(* Logix 5000 project; controller Receptivo vendor 1 type 14 code 106 rev 30.11; software revision 30.00; part 10 of 10 *)
(* tags used below, declared in another part *)
   CHASSIS_CURRENT : INT;
   CONTROLLER_STATUS : DINT;
   CPUdiag_FlashingGreen : BOOL;
   CPUdiag_FlashingRed : BOOL;
   CPUdiag_LEDStatus : DINT;
   CPUdiag_Major : MajorFaultBits;
   CPUdiag_MajorEvents : INT;
   CPUdiag_MajorFaultBits : DINT;
   CPUdiag_Minor : MinorFaultBits;
   CPUdiag_MinorEvents : INT;
   CPUdiag_MinorFaultBits : DINT;
   CPUdiag_SolidGreen : BOOL;
   CPUdiag_StatusMasked : INT;
   CPUdiag_StatusRaw : INT;
   INDEX : INT;
   IO_TREE_NO_OK : BOOL;
   IO_TREE_OK : DINT;
   MINOR_FAULTS : DINT;
   MODULE_MASK : DINT[10,17];
   MODULE_STATUS : DINT[10,17];
   Printer_Zebra_OK : BOOL;
   Timer1 : TIMER;
   ACTIVE_SLOT : DINT[10];
   Autonegotiation_Fallo : BOOL;
   Autonegotiation_OK : BOOL;
   Autonegotiation_Start : BOOL;
   AutoNegotiation_Status : SINT;
   CLOCK : DINT[7];
   Ethernet_Duplex_OK : BOOL;
   Ethernet_Duplex_State : ALIAS FOR Ethernet_Module_Status.1;
   Ethernet_Hardware_Mal : BOOL;
   Ethernet_Hardware_Status : ALIAS FOR Ethernet_Module_Status.6;
   Ethernet_Link_State : ALIAS FOR Ethernet_Module_Status.0;
   Ethernet_Module_Status : DINT;
   ETHERNET_STATUS : Ethernet_Status;
   FLASH_TIMERS : TIMER[2];
   FORCE_STATUS : DINT;
   Get_Ethernet_Module_Link_Status : MESSAGE;
   Hardy_Basculas_Net_OK : BOOL;
   KEY_SWITCH_REM_RUN : BOOL;
   KEY_SWITCH_RUN : BOOL;
   MODULE_FAULT_STATUS : DINT[10];
   Modulo_Ethernet_Mal : BOOL;
   Prueba : UDT_COLA[3];
   SYSTEM_STATUS_COMPLETE : BOOL;
   Velocidad_Modo_Forzado : BOOL;
(* SYSTEM_STATUS, continued *)

ROUTINE Ethernet_Module_Status   (* ladder *)
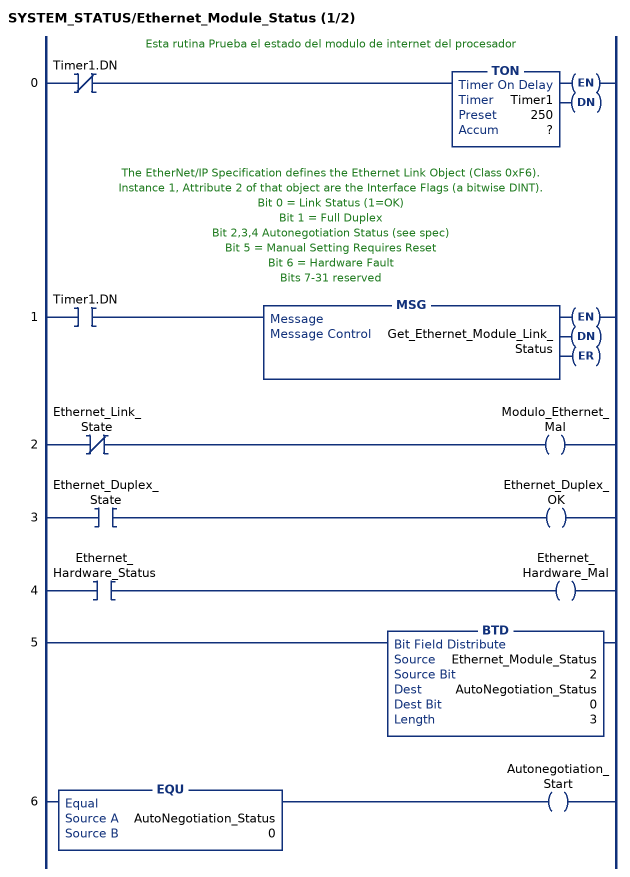
   // Esta rutina Prueba el estado del modulo de internet del procesador
   0: XIO(Timer1.DN)TON(Timer1,?,?);
   // The EtherNet/IP Specification defines the Ethernet Link Object (Class 0xF6).
   // Instance 1, Attribute 2 of that object are the Interface Flags (a bitwise DINT).
   // Bit 0 = Link Status (1=OK)
   // Bit 1 = Full Duplex
   // Bit 2,3,4 Autonegotiation Status (see spec)
   // Bit 5 = Manual Setting Requires Reset
   // Bit 6 = Hardware Fault
   // Bits 7-31 reserved
   1: XIC(Timer1.DN)MSG(Get_Ethernet_Module_Link_Status);
   2: XIO(Ethernet_Link_State)OTE(Modulo_Ethernet_Mal);
   3: XIC(Ethernet_Duplex_State)OTE(Ethernet_Duplex_OK);
   4: XIC(Ethernet_Hardware_Status)OTE(Ethernet_Hardware_Mal);
   5: BTD(Ethernet_Module_Status,2,AutoNegotiation_Status,0,3);
   6: EQU(AutoNegotiation_Status,0)OTE(Autonegotiation_Start);
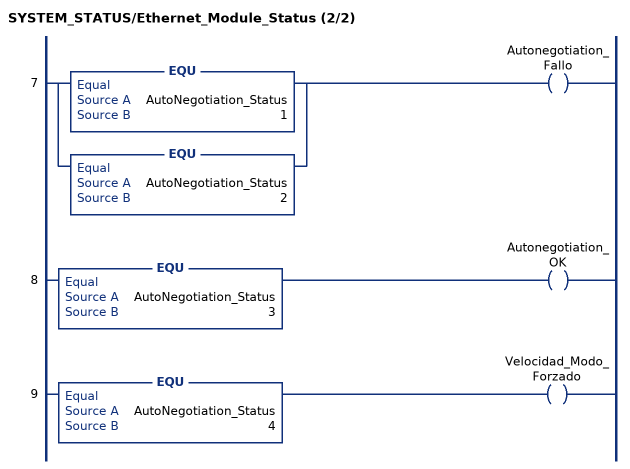
   7: [EQU(AutoNegotiation_Status,1) ,EQU(AutoNegotiation_Status,2) ]OTE(Autonegotiation_Fallo);
   8: EQU(AutoNegotiation_Status,3)OTE(Autonegotiation_OK);
   9: EQU(AutoNegotiation_Status,4)OTE(Velocidad_Modo_Forzado);
END_ROUTINE

ROUTINE ETHERNET_STATUS   (* ladder *)
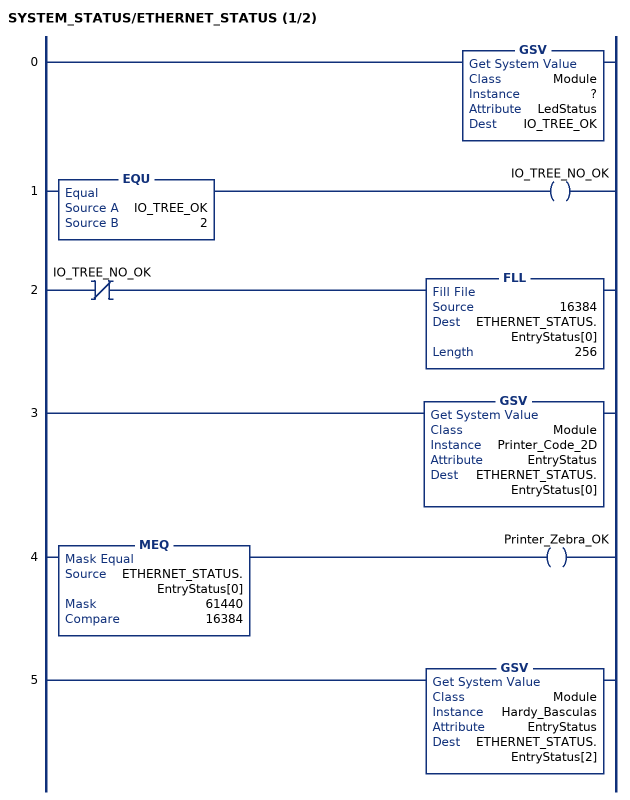
   0: GSV(Module,?,LedStatus,IO_TREE_OK);
   1: EQU(IO_TREE_OK,2)OTE(IO_TREE_NO_OK);
   2: XIO(IO_TREE_NO_OK)FLL(16384,ETHERNET_STATUS.EntryStatus[0],256);
   3: GSV(Module,Printer_Code_2D,EntryStatus,ETHERNET_STATUS.EntryStatus[0]);
   4: MEQ(ETHERNET_STATUS.EntryStatus[0],61440,16384)OTE(Printer_Zebra_OK);
   5: GSV(Module,Hardy_Basculas,EntryStatus,ETHERNET_STATUS.EntryStatus[2]);
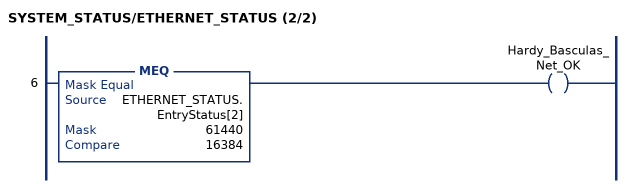
   6: MEQ(ETHERNET_STATUS.EntryStatus[2],61440,16384)OTE(Hardy_Basculas_Net_OK);
END_ROUTINE

ROUTINE GET_CONTROLLER_STATUS   (* ladder *)
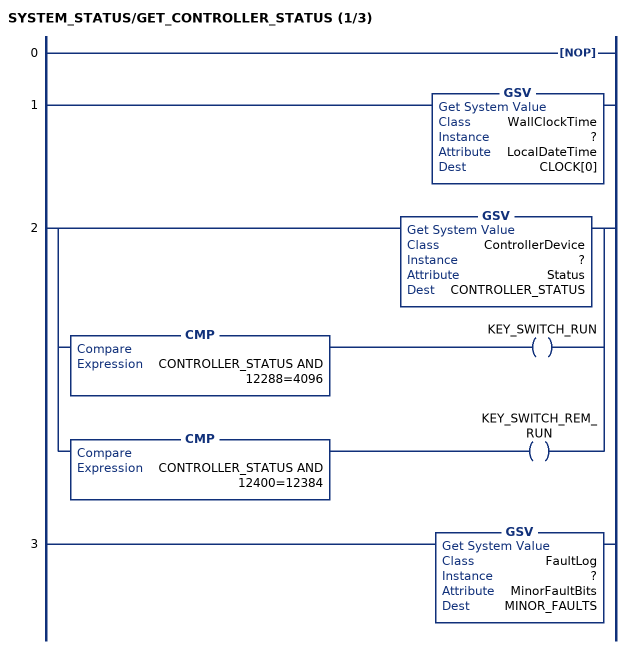
   0: NOP();
   1: GSV(WallClockTime,?,LocalDateTime,CLOCK[0]);
   2: [GSV(ControllerDevice,?,Status,CONTROLLER_STATUS) ,CMP(CONTROLLER_STATUS AND 12288=4096) OTE(KEY_SWITCH_RUN) ,CMP(CONTROLLER_STATUS AND 12400=12384) OTE(KEY_SWITCH_REM_RUN) ];
   3: GSV(FaultLog,?,MinorFaultBits,MINOR_FAULTS);
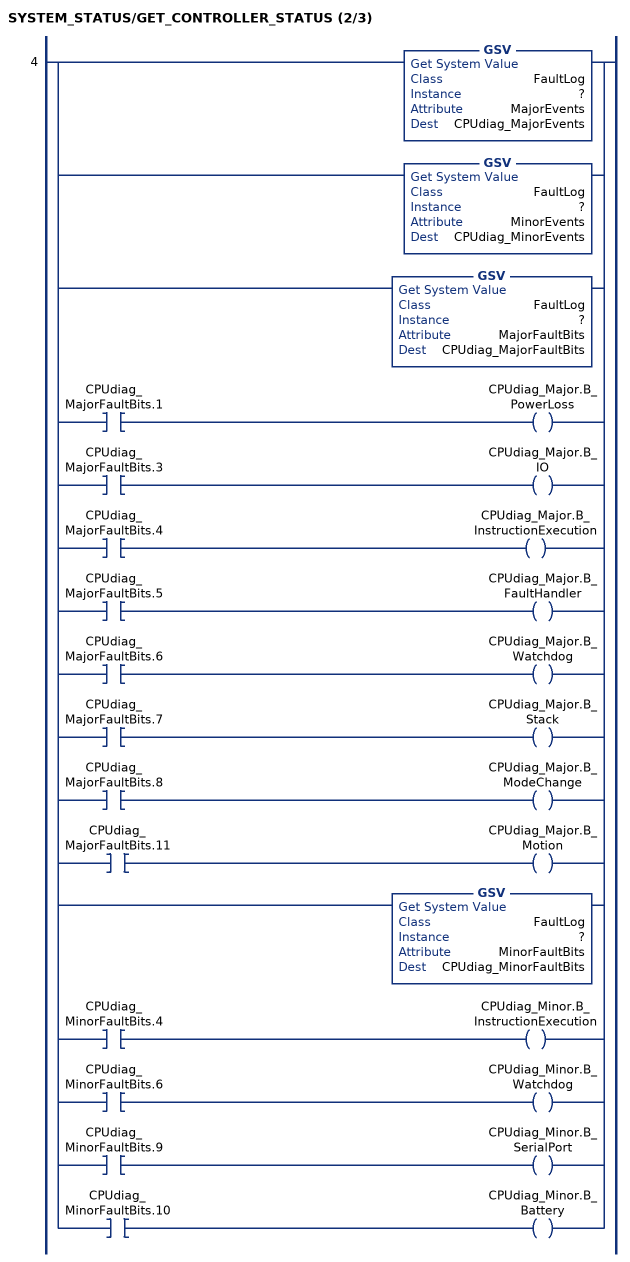
   4: [GSV(FaultLog,?,MajorEvents,CPUdiag_MajorEvents) ,GSV(FaultLog,?,MinorEvents,CPUdiag_MinorEvents) ,GSV(FaultLog,?,MajorFaultBits,CPUdiag_MajorFaultBits) ,XIC(CPUdiag_MajorFaultBits.1) OTE(CPUdiag_Major.B_PowerLoss) ,XIC(CPUdiag_MajorFaultBits.3) OTE(CPUdiag_Major.B_IO) ,XIC(CPUdiag_MajorFaultBits.4) OTE(CPUdiag_Major.B_InstructionExecution) ,XIC(CPUdiag_MajorFaultBits.5) OTE(CPUdiag_Major.B_FaultHandler) ,XIC(CPUdiag_MajorFaultBits.6) OTE(CPUdiag_Major.B_Watchdog) ,XIC(CPUdiag_MajorFaultBits.7) OTE(CPUdiag_Major.B_Stack) ,XIC(CPUdiag_MajorFaultBits.8) OTE(CPUdiag_Major.B_ModeChange) ,XIC(CPUdiag_MajorFaultBits.11) OTE(CPUdiag_Major.B_Motion) ,GSV(FaultLog,?,MinorFaultBits,CPUdiag_MinorFaultBits) ,XIC(CPUdiag_MinorFaultBits.4) OTE(CPUdiag_Minor.B_InstructionExecution) ,XIC(CPUdiag_MinorFaultBits.6) OTE(CPUdiag_Minor.B_Watchdog) ,XIC(CPUdiag_MinorFaultBits.9) OTE(CPUdiag_Minor.B_SerialPort) ,XIC(CPUdiag_MinorFaultBits.10) OTE(CPUdiag_Minor.B_Battery) ];
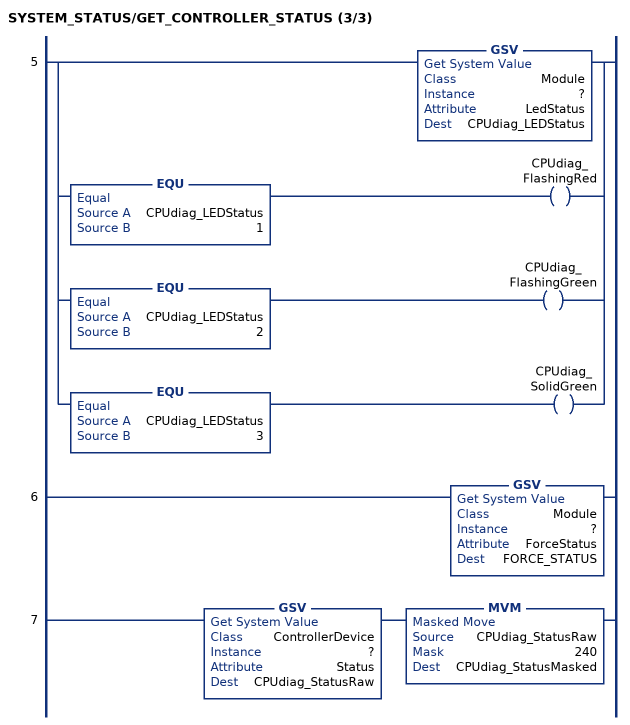
   5: [GSV(Module,?,LedStatus,CPUdiag_LEDStatus) ,EQU(CPUdiag_LEDStatus,1) OTE(CPUdiag_FlashingRed) ,EQU(CPUdiag_LEDStatus,2) OTE(CPUdiag_FlashingGreen) ,EQU(CPUdiag_LEDStatus,3) OTE(CPUdiag_SolidGreen) ];
   6: GSV(Module,?,ForceStatus,FORCE_STATUS);
   7: GSV(ControllerDevice,?,Status,CPUdiag_StatusRaw)MVM(CPUdiag_StatusRaw,240,CPUdiag_StatusMasked);
END_ROUTINE

ROUTINE GET_MODULE_STATUS   (* ladder *)
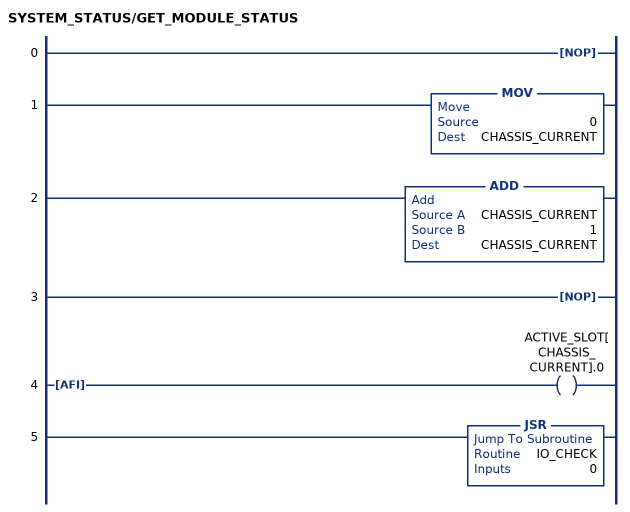
   0: NOP();
   1: MOV(0,CHASSIS_CURRENT);
   2: ADD(CHASSIS_CURRENT,1,CHASSIS_CURRENT);
   3: NOP();
   4: AFI()OTE(ACTIVE_SLOT[CHASSIS_CURRENT].0);
   5: JSR(IO_CHECK,0);
END_ROUTINE

ROUTINE IO_CHECK   (* ladder *)
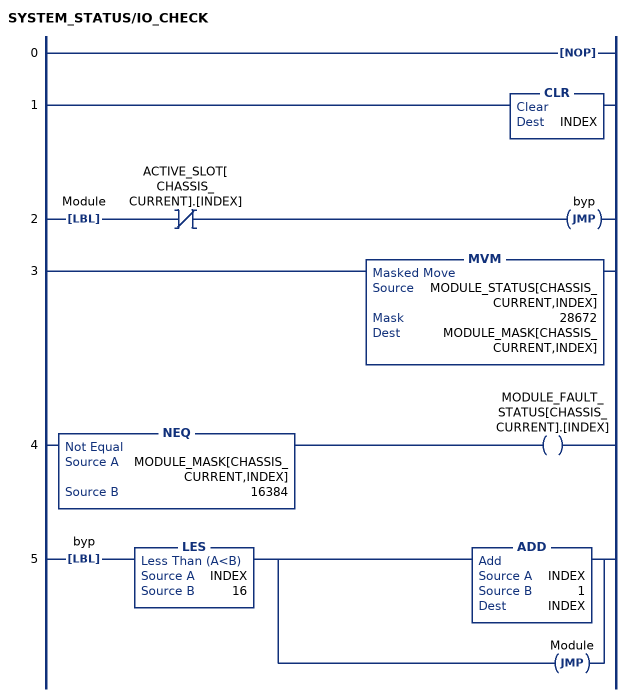
   0: NOP();
   1: CLR(INDEX);
   2: LBL(Module)XIO(ACTIVE_SLOT[CHASSIS_CURRENT].[INDEX])JMP(byp);
   3: MVM(MODULE_STATUS[CHASSIS_CURRENT,INDEX],28672,MODULE_MASK[CHASSIS_CURRENT,INDEX]);
   4: NEQ(MODULE_MASK[CHASSIS_CURRENT,INDEX],16384)OTE(MODULE_FAULT_STATUS[CHASSIS_CURRENT].[INDEX]);
   5: LBL(byp)LES(INDEX,16)[ADD(INDEX,1,INDEX) ,JMP(Module) ];
END_ROUTINE

ROUTINE MAIN   (* ladder *)
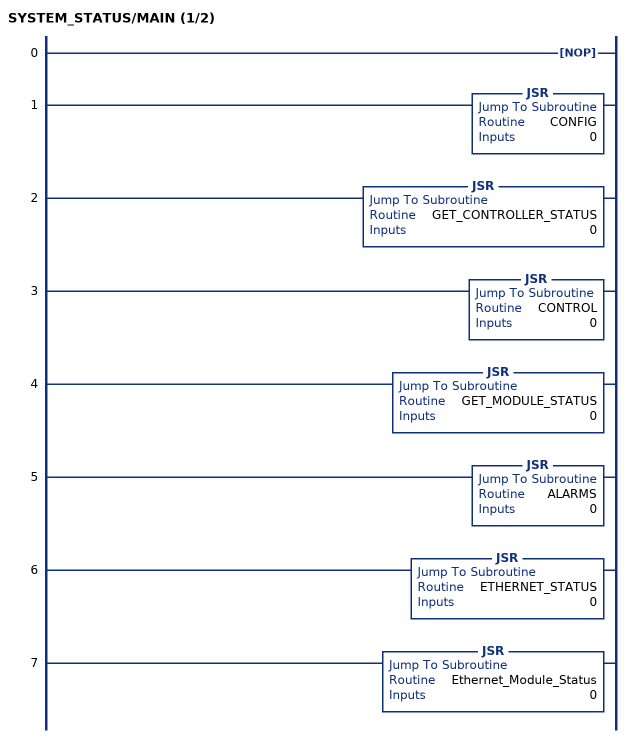
   0: NOP();
   1: JSR(CONFIG,0);
   2: JSR(GET_CONTROLLER_STATUS,0);
   3: JSR(CONTROL,0);
   4: JSR(GET_MODULE_STATUS,0);
   5: JSR(ALARMS,0);
   6: JSR(ETHERNET_STATUS,0);
   7: JSR(Ethernet_Module_Status,0);
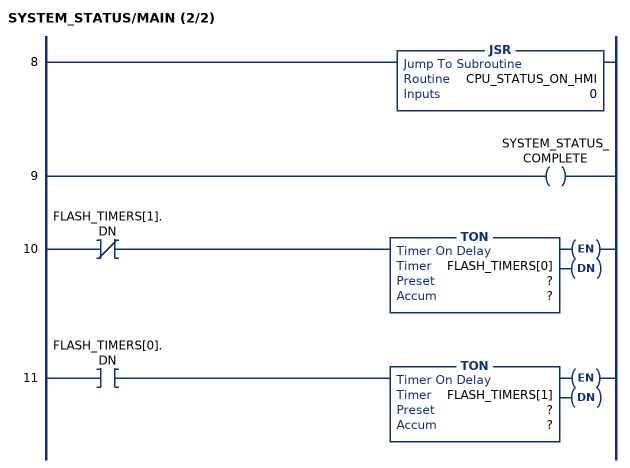
   8: JSR(CPU_STATUS_ON_HMI,0);
   9: OTE(SYSTEM_STATUS_COMPLETE);
   10: XIO(FLASH_TIMERS[1].DN)TON(FLASH_TIMERS[0],?,?);
   11: XIC(FLASH_TIMERS[0].DN)TON(FLASH_TIMERS[1],?,?);
END_ROUTINE
END_PROGRAM
